FUNCTION_BLOCK Sampling



VAR_INPUT
	S_start  :BOOL;//采集触发条件
	S_amount :UINT:=3;//采集次数
	S_site   :REAL ;//采集地址
	S_time   :REAL;//采集时间间隔
END_VAR

VAR_IN_OUT
	S_finish :BOOL;//采集完成	
END_VAR

VAR_OUTPUT
	Result_mean :REAL;//平均值
END_VAR




VAR
	a :UINT:=1;
	Sam_sum :REAL;//采样总值
	Sam_max :REAL;//采样最大值
	Sam_min :REAL;//采样最小值
	Cache_data :ARRAY[1..36000] OF  REAL;
	Sam_step :UINT;
	Sam_ton :Tc2_Standard.TON;
	S_time1 :TIME;
	Out_max :REAL;
END_VAR

S_time1:=REAL_TO_TIME(S_time*1000);
Sam_ton(PT:=S_time1);

IF S_amount>36000 THEN
	S_amount:=36000;
END_IF



CASE Sam_step OF
0:
IF 	S_start AND NOT S_finish THEN
	Result_mean:=0;
	a:=1;
	Sam_sum:=0;
	MEMSET(ADR(Cache_data),0,SIZEOF(Cache_data));
	Sam_step:=10;
END_IF

10:
IF a=(S_amount+1) THEN
	Sam_step:=500;
	ELSIF a<(S_amount+1) THEN
	Sam_step:=100;
END_IF

100:
Cache_data[a]:=S_site;
Sam_ton.IN:=TRUE;
Sam_step:=105;

105:
IF a=1 THEN
Sam_max:=Cache_data[a];	
Sam_min:=Cache_data[a];
Sam_step:=110;	
ELSE
Sam_step:=110;
END_IF


110:
IF Sam_ton.Q THEN
	Sam_step:=120;
	Sam_ton.IN:=FALSE;
END_IF

120:
IF Sam_max<Cache_data[a] THEN
	Sam_max:=Cache_data[a];
	Sam_step:=130;
	ELSE
	Sam_step:=130;
END_IF

130:

IF Sam_min>Cache_data[a] THEN
	Sam_min:=Cache_data[a];
	Sam_step:=140;
	ELSE
	Sam_step:=140;
END_IF


140:
Sam_sum:=Sam_sum+Cache_data[a];
a:=a+1;
Sam_step:=150;

150:
Sam_step:=10;

500:
Sam_sum:=(Sam_sum-Sam_max-Sam_min);
Sam_step:=510;

510:
Result_mean:=Sam_sum/(a-3);
S_finish:=TRUE;
Sam_step:=0;





END_CASE

END_FUNCTION_BLOCK

(* stored: Version 1.1.0.1, ProductVersion 3.1.4024.9
   POU Sampling: Id {9fb660dd-7ae2-4bf8-83e1-86b57cb64c78}, SpecialFunc None *)
